VAR_INPUT CONSTANT PERSISTENT				
	fHys 					: REAL;				// constant light: hysteresis for control-deviation. Limited from 0 to rBrtns
	{attribute 'parameterUnit':= 'ms'}          
	nSwiOvrTi				: UDINT;			// distinction time [ms] between short click and long-press
	{attribute 'parameterUnit':= 's'}       	
	nSwiTi					: UDINT;			// switch-ramp-time [s] to drive rOut from 0 to 100 
	{attribute 'parameterUnit':= 's'}       	
	nDimTi					: UDINT;			// dim-ramp-time [s] to drive rOut from 0 to 100 
	{attribute 'parameterUnit':= 's'}       	
	nRampTi					: UDINT;			// constant light: control-ramp-time [s]
	{attribute 'parameterUnit':= 's'}           
	nPreOffRampTi			: UDINT;			// ramp time [s] for the pre-off-function
	{attribute 'parameterUnit':= 's'}       	
	nBrtnsAdjTi				: UDINT;			// constant light: time [s] to let the brighness sensor adjust to new values before taking them over to the internal control
	{attribute 'parameterUnit':= '%'}           
	fOnValCtrl				: REAL;				// on value in control mode, limited from 0 to 100.
	{attribute 'parameterUnit':= '%'}           
	fOnValMan				: REAL;				// on value in memory mode, limited from 0 to 100.
	{attribute 'parameterUnit':= '%'}           
	fPreOffVal				: REAL;				// light value on pre-off-delay period.
	{attribute 'parameterUnit':= 's'}           
	nPreOffDly				: UDINT;			// duration [s] of pre-off-delay period
	{attribute 'parameterUnit':= '%'}           
	fMinVal 				: REAL;				// constant light: minimum control-value before the light control wants to turn off
	{attribute 'parameterUnit':= 's'}           
	nMinOffDly 				: UDINT;			// constant light: time [s] before switching off at fMinVal
	{attribute 'parameterUnit':= 's'}           
	nMinOnDly 				: UDINT;			// constant light: time [s] before switching on at fMinVal
	bMemoryMode				: BOOL;				// memory mode. switch on to value before last off	
	{attribute 'parameterUnit':= 'KELVIN'}	                    
	fLgtT					: REAL		:= 3000;	
END_VAR	
		             
VAR_INPUT CONSTANT           	
	SpBrightness			: FB_BA_AV_Op;
	ManMode					: FB_BA_LightingEvt :=( ePrio:= E_BA_LightingPrio.eManual);	
	CnstLgtAuto				: FB_BA_LightingEvt :=( ePrio:= E_BA_LightingPrio.eAutomaticLight);
END_VAR
VAR
	ConstLgtCtrl			: FB_BA_LightCtrlConst;	
	PrioSwi					: FB_BA_LightingTgmSel4;	
END_VAR

// call of external control (e.g. HMI)
SUPER^(); // FB_BA_Ext_LightConstCtrl
SpBrightness(); // FB_BA_AV_Op
ConstLgtCtrl(
    bSwi := bManualSwitch,
    bSwiUp := FALSE,
    bSwiDwn := FALSE,
    bOn := bOn,
    bOff := bOff,
    fSetValMan := fSetLightValueMan_In,
    bSetValMan := bSetLightValueMan_In,
    bSetCtrlMod := bSetCtrlMod_In,
    bRstManMod := FALSE,
    bRst := bResetRoomFunction,
    bPrc := bPresence,
    fBrtns := fBrightness,
    fSP := SpBrightness.fPresentValue,
    fHys := fHys,
    nSwiOvrTi := nSwiOvrTi,
    nSwiTi := nSwiTi,
    nDimTi := nDimTi,
    nRampTi := nRampTi,
    nPreOffRampTi := nPreOffRampTi,
    nBrtnsAdjTi := nBrtnsAdjTi,
    fOnValCtrl := fOnValCtrl,
    fOnValMan := fOnValMan,
    fPreOffVal := fPreOffVal,
    nPreOffDly := nPreOffDly,
    fMinVal := fMinVal,
    nMinOffDly := nMinOffDly,
    nMinOnDly := nMinOnDly,
    bMemMod := bMemoryMode,
    eLgtActMod := eLightActivationMode_In,
    fRefLgtVal := stReferenceFeedback.fLightValue); // FB_BA_LightCtrlConst
CnstLgtAuto(bEn := ConstLgtCtrl.bControlMode, fLgtVal := ConstLgtCtrl.fOut, fLgtT := fLgtT); // FB_BA_LightingEvt
ManMode(bEn := ConstLgtCtrl.bManualMode, fLgtVal := ConstLgtCtrl.fOut, fLgtT := fLgtT); // FB_BA_LightingEvt
bAdjusting := ConstLgtCtrl.bAdjusting;
PrioSwi(
    stLightingTgm_1 := CnstLgtAuto.stLighting,
    stLightingTgm_2 := ManMode.stLighting,
    stLightingTgm_3 := stAreaLighting,
    stLightingTgm_4 := stScene); // FB_BA_LightingTgmSel4
stLighting := PrioSwi.stLighting;
eActualPrio_Out := PrioSwi.ePrioActvTgm;
fLightValue_Out := stReferenceFeedback.fLightValue;
// information to external control (e.g. HMI)
bLightOn_Out := stReferenceFeedback.fLightValue > 0;
bErr_Out := stReferenceFeedback.bErr;
bCtrlMod_Out := ConstLgtCtrl.bControlMode;
// Reset external control commands
bSetLightValueMan_In := FALSE;
bSetCtrlMod_In := FALSE;

METHOD FB_init : BOOL
VAR_INPUT
	bInitRetains : BOOL; // if TRUE, the retain variables are initialized (warm start / cold start)
	bInCopyCode : BOOL;  // if TRUE, the instance afterwards gets moved into the copy code (online change)
END_VAR
SpBrightness.iParent		:= THIS^;
SpBrightness.iLabel			:= LblFun_Setpoint;
SpBrightness.eUnit			:= E_BA_Unit.eLight_Luxes;  
SpBrightness.fValueRm		:= 300.0;
SpBrightness.fCOVIncrement	:= BA2_Param.fDefCOVIncrement;	

fHys 						:= 50;		// constant-light: hysteresis for control-deviation [lux].
nSwiOvrTi					:= 250;		// distinction-time [ms] between short-lick and long-press
nSwiTi						:= 2;		// switch-ramp-time [s] to drive rOut from 0 to 100 
nDimTi						:= 10;		// dim-ramp-time [s] to drive rOut from 0 to 100 
nRampTi						:= 60;		// constant-light: control-ramp-time [s]
nPreOffRampTi				:= 2;		// ramp-time [s] for the pre-off-function
nBrtnsAdjTi					:= 5;		// constant-light: time [s] to let the brighness-sensor adjust to new values before taking them over to the internal control
fOnValCtrl					:= 50;		// on-Value, limited from 0 to 100.
fOnValMan					:= 100;		// on-Value, limited from 0 to 100.
fPreOffVal					:= 4;		// light-value on pre-off-delay period.
nPreOffDly					:= 10;		// duration [s] of pre-off-delay period
fMinVal 					:= 4;		// constant-light: minimum control-value before the light control wants to turn off
nMinOffDly 					:= 300;		// constant-light: time [s] before switching off at fMinVal
nMinOnDly 					:= 300;		// constant-light: time [s] before switching on at fMinVal
bMemoryMode					:= FALSE;	// memory-mode. switch on to value before last off

fLgtT						:= 3000;			// [K]
END_METHOD

END_FUNCTION_BLOCK

// ---- Templates/POUs/Trade/RoomAutomation/Lighting/[Internal]/FB_BA_Ext_LightConstCtrl.TcPOU
{region '#Template'}
	{attribute 'Version' := '5.0.0.0'}
	{attribute 'Tags' := '"LCID": "1031", "Text": "RA, Beleuchtung, Anwenderfunktionen, Zone"'}
	{attribute 'Tags' := '"LCID": "1033", "Text": "RA, Lighting, User-functions, zone"'}
	{attribute 'Using' := '"Type": "Template", "URI": "ST_BA_LightActuatorFeedback"'}
	{attribute 'Description' := '"LCID": "1031", "Text": "Beleuchtung interner Baustein"'}
	{attribute 'Description' := '"LCID": "1033", "Text": "Lighting internal function"'}
{endregion}
FUNCTION_BLOCK FB_BA_Ext_LightConstCtrl EXTENDS FB_BA_Ext_LightCtrl
VAR	
	// data from/to user function
	{attribute 'BaParam.Title.DE' := 'Aktivieren Regelungsbetrieb'}
	{attribute 'BaParam.Title.EN' := 'Activate control mode'}
	{attribute 'BaParam.Access.Write' := 'Basic'}
	bSetCtrlMod_In				: BOOL;						// enter control mode from either deactivated or manual mode
	{attribute 'BaParam.Title.DE' := 'Regelungsbetrieb ist aktiv'}
	{attribute 'BaParam.Title.EN' := 'Control mode is active'}
	{attribute 'BaParam.Access.Write' := 'Locked'}
	{attribute 'BaParam.Access.Read' := 'Guest'}
	bCtrlMod_Out				: BOOL;						// state information control mode, used for external display
END_VAR

SUPER^();

END_FUNCTION_BLOCK

// ---- Templates/POUs/Trade/RoomAutomation/RoomSamples/FB_BA_RoomSample1.TcPOU
{region '#Template'}
	{attribute 'Version' := '6.0.0.0'}
	{attribute 'Tags' := '"LCID": "1031", "Text": "RA, Room, Sample"'}
	{attribute 'Tags' := '"LCID": "1033", "Text": "RA, Room, Sample"'}
	{attribute 'Using' := '"Type": "Template", "URI": "Site"'}
	{attribute 'Using' := '"Type": "Template", "URI": "BA2_Param"'}
	{attribute 'Using' := '"Type": "Template", "URI": "ST_BA_Facade"'}
	{attribute 'Using' := '"Type": "Template", "URI": "ST_BA_Lighting"'}
	{attribute 'Description' := '"LCID": "1031", "Text": "Beispiel Template Raum"'}
	{attribute 'Description' := '"LCID": "1033", "Text": "Sample-template room"'}
{endregion}
FUNCTION_BLOCK FB_BA_RoomSample1 EXTENDS FB_BA_View
VAR_INPUT
	stFacade					: ST_BA_Facade;			// sunblind-data from the next higher level
	stAreaLighting				: ST_BA_Lighting;		// lighting-data from the next higher level
END_VAR
		
VAR_INPUT CONSTANT PERSISTENT					
	{attribute 'parameterUnit':= 'KELVIN'}	                    
	fRmTAdjMin					: REAL;
	{attribute 'parameterUnit':= 'KELVIN'}	                    
	fRmTAdjMax					: REAL;
	{attribute 'parameterUnit':= 'KELVIN'}	                    
	fLgtT						: REAL;
	{attribute 'parameterUnit':= 's'}	                    
	nPollingIntervalFast		: UDINT;
	{attribute 'parameterUnit':= 's'}	                    
	nPollingIntervalNormal		: UDINT;
END_VAR	

VAR_INPUT CONSTANT
	BrtnsPrcSns					: FB_BA_BrightnessPresenceDALI;
	                    		
	Ctrl						: FB_BA_HeatCool_PID;
	VlvHtg						: FB_BA_ActuatorAnalog;
 	VlvCol						: FB_BA_ActuatorAnalog;
	                    		
	WdwCon1						: FB_BA_SensorBinary;
	WdwCon2						: FB_BA_SensorBinary;
	DewPointSensor				: FB_BA_SensorBinary;	
	RmTSen						: FB_BA_SensorAnalog;
	RmTAdj						: FB_BA_SensorAnalog;
	SunBldZone					: FB_BA_SunblindZone;
	SunBld1						: FB_BA_SunBld;		
	SunBld2						: FB_BA_SunBld;				
	LightZoneConstant			: FB_BA_LightGroupConstant;
	Light1						: FB_BA_LightAnalog;
	Light2						: FB_BA_LightAnalog;
END_VAR                 		
VAR                     		
	bSunbldSwiUp				: BOOL;
	bSunbldSwiDwn				: BOOL;	
	bLightSwi					: BOOL;	
	RmTAvg						: FB_BA_EnAvrg02;
	bInitializeSensor			: BOOL;	
END_VAR
VAR // added by the converter: edge detectors and wires of the graphical bodies
    _s1, _s2 : ST_BA_Analog;
END_VAR

SUPER^(); // FB_BA_View
BrtnsPrcSns(
    bEn := TRUE,
    bInitialize := bInitializeSensor,
    nPrdQueryBrtns := SEL(LightZoneConstant.bAdjusting, nPollingIntervalNormal, nPollingIntervalFast)); // FB_BA_BrightnessPresenceDALI
bInitializeSensor := FALSE;
WdwCon1(); // FB_BA_SensorBinary
WdwCon2(); // FB_BA_SensorBinary
DewPointSensor(); // FB_BA_SensorBinary
RmTSen(); // FB_BA_SensorAnalog
RmTAdj(); // FB_BA_SensorAnalog
Ctrl(
    bPrc := BrtnsPrcSns.bPresence,
    bWdwCon := NOT WdwCon1.bPresentValue OR NOT WdwCon2.bPresentValue,
    eMedium := Site.eHeatCoolMedium,
    bDewPnt := NOT DewPointSensor.bPresentValue,
    fRmT := RmTSen.fPresentValue,
    fRmTAdj := LIMIT(fRmTAdjMin, RmTAdj.fPresentValue, fRmTAdjMax),
    stBuildingSpRmT := Site.stBuildingSpRmT,
    eBuildingEnergyLevel := Site.eBuildingEnergyLevel); // FB_BA_HeatCool_PID
// compose _s1 : ST_BA_Analog
_s1.bEnPgm := Ctrl.bCtrlHtgActv;
_s1.fValPgm := Ctrl.fCtrlValHtg;
VlvHtg(stCmd := _s1); // FB_BA_ActuatorAnalog
// compose _s2 : ST_BA_Analog
_s2.bEnPgm := Ctrl.bCtrlColActv;
_s2.fValPgm := Ctrl.fCtrlValCol;
VlvCol(stCmd := _s2); // FB_BA_ActuatorAnalog
SunBldZone(
    fRoomTempSen := RmTAvg.fAvgVal,
    bPrcDetc := BrtnsPrcSns.bPresence,
    bSwiUp := bSunbldSwiUp,
    bSwiDwn := bSunbldSwiDwn,
    bRstManFnct := BrtnsPrcSns.bRstSwi,
    stBuildingSpRmT := Site.stBuildingSpRmT,
    stFacade := stFacade,
    stReferenceFeedback := SunBld1.stFeedback); // FB_BA_SunblindZone
SunBld2(bEn := TRUE, stSunBldCmd := SunBldZone.stSunBldOut); // FB_BA_SunBld
SunBld1(bEn := TRUE, stSunBldCmd := SunBldZone.stSunBldOut); // FB_BA_SunBld
LightZoneConstant(
    bManualSwitch := bLightSwi,
    bOn := FALSE,
    bOff := FALSE,
    bResetRoomFunction := BrtnsPrcSns.bRstSwi,
    bPresence := BrtnsPrcSns.bPresence,
    fBrightness := BrtnsPrcSns.fBrightness,
    stAreaLighting := stAreaLighting,
    stReferenceFeedback := Light1.stFeedback); // FB_BA_LightGroupConstant
Light2(bEn := TRUE, stLightingCmd := LightZoneConstant.stLighting); // FB_BA_LightAnalog
Light1(bEn := TRUE, stLightingCmd := LightZoneConstant.stLighting); // FB_BA_LightAnalog

METHOD FB_init : BOOL
VAR_INPUT
	bInitRetains : BOOL; // if TRUE, the retain variables are initialized (warm start / cold start)
	bInCopyCode : BOOL;  // if TRUE, the instance afterwards gets moved into the copy code (online change)
END_VAR
BrtnsPrcSns.iParent							:= THIS^;
BrtnsPrcSns.iLabel							:= LblCtl_BrightnessPresenceSensor; 			
BrtnsPrcSns.eDPADMode						:= E_BA_DPADMode.eInclude;	
BrtnsPrcSns.nAdr							:= 11;
BrtnsPrcSns.nInstancePresence				:= 1;	
BrtnsPrcSns.nInstanceBrightness				:= 0;
BrtnsPrcSns.nResBrtns						:= 10;
BrtnsPrcSns.ipDALICommunication				:= DALICommunication.fbKL6821Communication;

nPollingIntervalFast						:= 1;			// fast interval polling the light-value e.g. in case of active light-adapting
nPollingIntervalNormal						:= 15;			// slow interval polling the light-value

WdwCon1.iParent								:= THIS^;
WdwCon1.iLabel								:= LblAgg_WindowContact; 			
WdwCon1.eDPADMode							:= E_BA_DPADMode.eInclude;		
WdwCon1.Input.iLabel						:= LblFun_Status; 	
WdwCon1.Input.ePolarity						:= E_BA_Polarity.eReverse;
WdwCon1.Input.sActiveText 					:= txtEvent_Closed;
WdwCon1.Input.sInactiveText 				:= txtEvent_Opened;
WdwCon1.Input.nEventClassID					:= EC_ID.NC50;
WdwCon1.Input.aEventTransitionText[1]		:= txtEvent_Disturb;
WdwCon1.Input.aEventTransitionText[2]		:= txtEvent_None;
WdwCon1.Input.aEventTransitionText[3]		:= txtEvent_Normal;
WdwCon1.Input.bEventDetectionEnable			:= FALSE;
                                    		
WdwCon2.iParent								:= THIS^;
WdwCon2.iLabel								:= LblAgg_WindowContact; 			
WdwCon2.eDPADMode							:= E_BA_DPADMode.eInclude;		
WdwCon2.Input.iLabel						:= LblFun_Status; 	
WdwCon2.Input.ePolarity						:= E_BA_Polarity.eReverse;
WdwCon2.Input.sActiveText 					:= txtEvent_Closed;
WdwCon2.Input.sInactiveText 				:= txtEvent_Opened;
WdwCon2.Input.nEventClassID					:= EC_ID.NC50;
WdwCon2.Input.aEventTransitionText[1]		:= txtEvent_Disturb;
WdwCon2.Input.aEventTransitionText[2]		:= txtEvent_None;
WdwCon2.Input.aEventTransitionText[3]		:= txtEvent_Normal;
WdwCon2.Input.bEventDetectionEnable			:= FALSE;

DewPointSensor.iParent						:= THIS^;
DewPointSensor.iLabel						:= LblAgg_MonitorDewPoint; 			
DewPointSensor.eDPADMode					:= E_BA_DPADMode.eInclude;		
DewPointSensor.Input.iLabel					:= LblFun_Status; 	
DewPointSensor.Input.ePolarity				:= E_BA_Polarity.eReverse;	
DewPointSensor.Input.sActiveText 			:= txtEvent_Normal;
DewPointSensor.Input.sInactiveText 			:= txtEvent_Triggered;
DewPointSensor.Input.nEventClassID			:= EC_ID.NC40;
DewPointSensor.Input.aEventTransitionText[1]:= txtEvent_Triggered;
DewPointSensor.Input.aEventTransitionText[2]:= txtEvent_None;
DewPointSensor.Input.aEventTransitionText[3]:= txtEvent_Normal;
DewPointSensor.Input.bEventDetectionEnable	:= TRUE;

RmTSen.iParent								:= THIS^;
RmTSen.iLabel								:= LblAgg_TemperatureRoomAir; 			
RmTSen.eDPADMode							:= E_BA_DPADMode.eInclude;		
RmTSen.MV.eUnit 							:= E_BA_Unit.eTemperature_DegreesCelsius;
RmTSen.MV.nEventClassID						:= EC_ID.NC60;
RmTSen.MV.aEventTransitionText[1]			:= txtEvent_Disturb;
RmTSen.MV.aEventTransitionText[2]			:= txtEvent_None;
RmTSen.MV.aEventTransitionText[3]			:= txtEvent_Normal;
RmTSen.MV.eEnPlantLock						:= E_BA_LockPriority.eNoLock;
RmTSen.MV.fResolution 						:= 0.01;
RmTSen.MV.fScaleOffset 						:= 0; 
                     			        	
RmTAdj.iParent								:= THIS^;
RmTAdj.iLabel								:= LblAgg_RoomControlUnit; 	
RmTAdj.eDPADMode							:= E_BA_DPADMode.eInclude;		
RmTAdj.MV.eUnit 							:= E_BA_Unit.eTemperature_DegreesKelvin;
RmTAdj.MV.nEventClassID						:= EC_ID.NC60;
RmTAdj.MV.aEventTransitionText[1]			:= txtEvent_Disturb;
RmTAdj.MV.aEventTransitionText[2]			:= txtEvent_None;
RmTAdj.MV.aEventTransitionText[3]			:= txtEvent_Normal;
RmTAdj.MV.eEnPlantLock						:= E_BA_LockPriority.eNoLock;
RmTAdj.MV.fResolution 						:= 0.01;
RmTAdj.MV.fScaleOffset 						:= 0; 
        
fRmTAdjMin									:= -5;	// limits of room-temperature-adjustment           
fRmTAdjMax									:= 5;	// in order to prevent adjusting from 0 to 50 degrees, for example

Ctrl.iParent								:= THIS^;
Ctrl.iLabel									:= LblCtl_RoomTemperatureControl; 			 
Ctrl.eDPADMode								:= E_BA_DPADMode.eInclude;

VlvHtg.iParent								:= THIS^;
VlvHtg.iLabel								:= LblAgg_Valve; 	
VlvHtg.eDPADMode							:= E_BA_DPADMode.eInclude;
VlvHtg.Mdlt.eUnit 							:= E_BA_Unit.eOther_Percent;
VlvHtg.Mdlt.nEventClassID					:= EC_ID.NC60;
VlvHtg.Mdlt.aEventTransitionText[1]			:= txtEvent_Disturb;
VlvHtg.Mdlt.aEventTransitionText[2]			:= txtEvent_None;
VlvHtg.Mdlt.aEventTransitionText[3]			:= txtEvent_Normal;		
VlvHtg.Mdlt.fResolution 					:= 0.01;
VlvHtg.Mdlt.fScaleOffset 					:= 0; 		 
                            			    
VlvCol.iParent								:= THIS^;
VlvCol.iLabel								:= LblAgg_Valve; 	
VlvCol.eDPADMode							:= E_BA_DPADMode.eInclude;
VlvCol.Mdlt.eUnit 							:= E_BA_Unit.eOther_Percent;
VlvCol.Mdlt.nEventClassID					:= EC_ID.NC60;
VlvCol.Mdlt.aEventTransitionText[1]			:= txtEvent_Disturb;
VlvCol.Mdlt.aEventTransitionText[2]			:= txtEvent_None;
VlvCol.Mdlt.aEventTransitionText[3]			:= txtEvent_Normal;		
VlvCol.Mdlt.fResolution 					:= 0.01;
VlvCol.Mdlt.fScaleOffset 					:= 0; 



SunBldZone.iParent							:= THIS^;
SunBldZone.iLabel							:= LblCtl_SunblindZoneControl; 		

Sunbld1.iParent								:= THIS^;
Sunbld1.iLabel								:= LblCtl_SunblindActuator; 	
Sunbld1.sObjectName							:= '{Idx=01}';		 		 
Sunbld1.eDPADMode							:= E_BA_DPADMode.eInclude;

Sunbld2.iParent								:= THIS^;
Sunbld2.iLabel								:= LblCtl_SunblindActuator; 	
Sunbld2.sObjectName							:= '{Idx=02}';	 		 
Sunbld2.eDPADMode							:= E_BA_DPADMode.eInclude;



Light1.iParent								:= THIS^;
Light1.iLabel								:= LblCtl_LightActuator; 	
Light1.sObjectName							:= '{Idx=01}';		 
Light1.eDPADMode							:= E_BA_DPADMode.eInclude;

Light2.iParent								:= THIS^;
Light2.iLabel								:= LblCtl_LightActuator; 		
Light2.sObjectName							:= '{Idx=02}';	 
Light2.eDPADMode							:= E_BA_DPADMode.eInclude;

LightZoneConstant.iParent					:= THIS^;
LightZoneConstant.iLabel					:= LblCtl_LightZoneControl; 			 
LightZoneConstant.eDPADMode					:= E_BA_DPADMode.eInclude;

fLgtT										:= 3000;		// light-temperature [K]
END_METHOD

END_FUNCTION_BLOCK

// ---- Templates/POUs/Trade/RoomAutomation/SunProtection/Actuators/FB_BA_SunBld.TcPOU
{region '#Template'}
	{attribute 'Version' := '6.0.0.0'}
	{attribute 'Tags' := '"LCID": "1031", "Text": "RA, Sunprotection, Sunblind"'}
	{attribute 'Tags' := '"LCID": "1033", "Text": "RA, Sunprotection, Sunblind"'}
	{attribute 'Using' := '"Type": "Template", "URI": "BA2_Param"'}
	{attribute 'Using' := '"Type": "Template", "URI": "ST_BA_SunblindActuatorFeedback"'}
	{attribute 'Description' := '"LCID": "1031", "Text": "Sonnenschutzaktor (Jalousie)"'}
	{attribute 'Description' := '"LCID": "1033", "Text": "Sunblind-actuator (venetian blind)"'}
{endregion}
FUNCTION_BLOCK FB_BA_SunBld EXTENDS FB_BA_View


VAR_INPUT
	bEn						: BOOL;
	stSunBldCmd				: ST_BA_SunBld;		// Low-Priorities command telegram
END_VAR
VAR_OUTPUT
	bReferencing			: BOOL;				// device is being referenced
	nReferenceTimer			: UDINT;            
	bErr					: BOOL;				// error
	fActualPosition			: REAL;				// actual position
	fActualAngle			: REAL;				// actual angle
	eActualSunblindPrio		: BYTE;				// actual telegram priority
	stFeedback				: ST_BA_SunblindActuatorFeedback;
END_VAR
VAR_INPUT CONSTANT PERSISTENT
	{attribute 'parameterUnit':= 'ms'}
	nPositioningDelay		: UDINT;	// delay of automatic telegrams [ms] to prevent overload
	{attribute 'parameterUnit':= 'ms'}  
	nTiUp					: UDINT;	// total driving-up-time [ms]
	{attribute 'parameterUnit':= 'ms'}  
	nTiDwn					: UDINT;	// total driving-down-time [ms]
	{attribute 'parameterUnit':= 'ms'}          		
	nTurnTiUp				: UDINT;	// time to turn lamellas up [ms]
	{attribute 'parameterUnit':= 'ms'}          		
	nTurnTiDwn				: UDINT;	// time to turn lamellas down [ms]
	{attribute 'parameterUnit':= 'ms'}          		
	nBckLshTiUp				: UDINT;	// Time to traverse the backlash in the upward direction [ms]
	{attribute 'parameterUnit':= 'ms'}          		
	nBckLshTiDwn			: UDINT;	// Time to traverse the backlash in the downward direction [ms]
	{attribute 'parameterUnit':= 'deg'} 
	fAnglLmtUp				: REAL;		// upper limit of lamellas in deg - must be greater than fAnglLmtDwn
	{attribute 'parameterUnit':= 'deg'} 
	fAnglLmtDwn				: REAL;		// lower limit of lamellas in deg - must be lower than fAnglLmtUp
END_VAR
VAR_INPUT CONSTANT				 
	ActualPosition			: FB_BA_AV_Op;		
	ActualAngle				: FB_BA_AV_Op;		
END_VAR
VAR
	PositioningDelay		: FB_BA_SunBldPosDly;
	SunBldActr				: FB_BA_SunBldActr;
	bCmdUp			AT %Q*	: BOOL;
	bCmdDown		AT %Q*	: BOOL;
END_VAR
VAR // added by the converter: edge detectors and wires of the graphical bodies
    _s1 : ST_BA_SunblindActuatorFeedback;
END_VAR

SUPER^(); // FB_BA_View
PositioningDelay(stIn := stSunBldCmd, nDly := nPositioningDelay); // FB_BA_SunBldPosDly
SunBldActr(
    bEn := bEn,
    stCmd := PositioningDelay.stOut,
    nTiUp := nTiUp,
    nTiDwn := nTiDwn,
    nTurnTiUp := nTurnTiUp,
    nTurnTiDwn := nTurnTiDwn,
    nBckLshTiUp := nBckLshTiUp,
    nBckLshTiDwn := nBckLshTiDwn,
    fAnglLmtUp := fAnglLmtUp,
    fAnglLmtDwn := fAnglLmtDwn); // FB_BA_SunBldActr
bCmdUp := SunBldActr.bUp;
bCmdDown := SunBldActr.bDwn;
fActualPosition := SunBldActr.fActlPos;
fActualAngle := SunBldActr.fActlAngl;
bReferencing := SunBldActr.bRef;
nReferenceTimer := SunBldActr.nRefTi;
bErr := SunBldActr.bErr;
ActualPosition(fValuePgm := fActualPosition); // FB_BA_AV_Op
ActualAngle(fValuePgm := fActualAngle); // FB_BA_AV_Op
eActualSunblindPrio := stSunBldCmd.ePrio;
// compose _s1 : ST_BA_SunblindActuatorFeedback
_s1.bReferencing := SunBldActr.bRef;
_s1.bErr := SunBldActr.bErr;
_s1.bBusy := SunBldActr.bBusy;
_s1.ePrio := stSunBldCmd.ePrio;
_s1.fPosition := SunBldActr.fActlPos;
_s1.fAngle := SunBldActr.fActlAngl;
_s1.fAnglLmtUp := fAnglLmtUp;
_s1.fAnglLmtDwn := fAnglLmtDwn;
stFeedback := _s1;

METHOD FB_init : BOOL
VAR_INPUT
	bInitRetains : BOOL; // if TRUE; the retain variables are initialized (warm start / cold start)
	bInCopyCode : BOOL;  // if TRUE; the instance afterwards gets moved into the copy code (online change)
END_VAR
nPositioningDelay				:= 250;			// delay of automatic telegrams [ms] to prevent overload
nTiUp							:= 50000;		// total driving-up-time [ms]
nTiDwn							:= 50000;		// total driving-down-time [ms]
nTurnTiUp						:= 1500;		// time to turn lamellas up [ms]
nTurnTiDwn						:= 1500;		// time to turn lamellas down [ms]
nBckLshTiUp						:= 100;			// Time to traverse the backlash in the upward direction [ms]
nBckLshTiDwn					:= 100;			// Time to traverse the backlash in the downward direction [ms]
fAnglLmtUp						:= 30;			// upper limit of lamellas in deg - must be greater than fAnglLmtDwn
fAnglLmtDwn						:= -70;			// lower limit of lamellas in deg - must be lower than fAnglLmtUp

// actual position / aktueller Position
ActualPosition.iParent			:= THIS^;
ActualPosition.iLabel			:= LblFun_FeedbackSunblindPosition;
ActualPosition.eUnit			:= E_BA_Unit.eOther_Percent;
ActualPosition.fCOVIncrement	:= BA2_Param.fDefCOVIncrement;

// actual angle / aktueller Lamellenwinkel
ActualAngle.iParent				:= THIS^;
ActualAngle.iLabel				:= LblFun_FeedbackSunblindAngle;
ActualAngle.eUnit				:= E_BA_Unit.eOther_DegreesAngular;
ActualAngle.fCOVIncrement		:= BA2_Param.fDefCOVIncrement;
END_METHOD

END_FUNCTION_BLOCK

// ---- Templates/POUs/Trade/RoomAutomation/SunProtection/[Internal]/FB_BA_Ext_SunblindBase.TcPOU
{region '#Template'}
	{attribute 'Version' := '5.0.0.0'}
	{attribute 'Tags' := '"LCID": "1031", "Text": "RA, Sunprotection, Sunblind, Zone"'}
	{attribute 'Tags' := '"LCID": "1033", "Text": "RA, Sunprotection, Sunblind, Zone"'}
	{attribute 'Using' := '"Type": "Template", "URI": "ST_BA_Facade"'}
	{attribute 'Description' := '"LCID": "1031", "Text": "Sonnenschutzlogik interner Baustein"'}
	{attribute 'Description' := '"LCID": "1033", "Text": "Sunblind-logic inernal function)"'}
{endregion}
FUNCTION_BLOCK FB_BA_Ext_SunblindBase EXTENDS FB_BA_Object
VAR_INPUT
	bRstManFnct				: BOOL;								// reset the external function from outside
END_VAR
VAR		
	{attribute 'BaParam.Title.DE' := 'Hoch'}
	{attribute 'BaParam.Title.EN' := 'Up'}
	{attribute 'BaParam.Access.Write' := 'Basic'}
	bUp_In					: BOOL;								// from external
	{attribute 'BaParam.Title.DE' := 'Herunter'}
	{attribute 'BaParam.Title.EN' := 'Down'}
	{attribute 'BaParam.Access.Write' := 'Basic'}
	bDown_In				: BOOL;								// from external
	{attribute 'BaParam.Title.DE' := 'Reset Hand'}
	{attribute 'BaParam.Title.EN' := 'Reset manual'}
	{attribute 'BaParam.Access.Write' := 'Basic'}
	bResetManual_In			: BOOL;								// from external
	{attribute 'BaParam.Title.DE' := 'Rückmeldung Fehler'}
	{attribute 'BaParam.Title.EN' := 'Feedback Error'}
	{attribute 'BaParam.Access.Write' := 'Locked'}
	{attribute 'BaParam.Access.Read' := 'Guest'}
	bErr_Out				: BOOL;								// to external
	{attribute 'BaParam.Title.DE' := 'Rückmeldung geöffnet'}
	{attribute 'BaParam.Title.EN' := 'Feedback open'}
	{attribute 'BaParam.Access.Write' := 'Locked'}
	{attribute 'BaParam.Access.Read' := 'Guest'}
	bOpened_Out				: BOOL;								// to external
	{attribute 'BaParam.Title.DE' := 'Rückmeldung geschlossen'}
	{attribute 'BaParam.Title.EN' := 'Feedback close'}
	{attribute 'BaParam.Access.Write' := 'Locked'}
	{attribute 'BaParam.Access.Read' := 'Guest'}
	bClosed_Out				: BOOL;								// to external
	{attribute 'BaParam.Title.DE' := 'Aktuell steuernde Priorität'}
	{attribute 'BaParam.Title.EN' := 'Actual controlling priority'}
	{attribute 'BaParam.Access.Write' := 'Locked'}
	{attribute 'BaParam.Access.Read' := 'Guest'}
	eActualPrio_Out			: BYTE;								// priority of resulting zone-telegram
		                                                    	
	                                                        	
	bInitialize_In			: BOOL;								// from external // actually not used by external control
	bBusy					: BOOL;								// to external // actually not used by external control
	bReferencing			: BOOL;								// to external // actually not used by external control
	bBlindMoving			: BOOL;                         	
	                                                        	
	stSunblindCmdExt		: ST_BA_SunBld;						// telegram assembled from external data
	stSunblindCmdResult		: ST_BA_SunBld;						// telegram to extract information for external handling
		                    
	rtUp					: R_TRIG;
	rtDown					: R_TRIG;
	rtReferencing			: R_TRIG;
	ftBusy					: F_TRIG;
	                        
	_nResetManual_In		: BYTE;
	_nInitialize_In			: BYTE;
END_VAR
VAR_INPUT CONSTANT PERSISTENT
	ePrio					: BYTE	:= E_BA_SunbldPrio.eManualGroup;	// priority of external telegram
END_VAR

SUPER^();

// predefinition of priority
stSunblindCmdExt.ePrio		:= ePrio;

// state moving
bBlindMoving	:= bBusy AND NOT bReferencing;

// reset telegram from outside or from HMI or set 0%/100% as on/off
IF bRstManFnct	OR (bResetManual_In AND (_nResetManual_In=1))	THEN	// bResetManual_In has to go through the other parts first before having an effect here
	stSunblindCmdExt.bActv			:= FALSE;
	stSunblindCmdExt.bManUp			:= FALSE;
	stSunblindCmdExt.bManDwn		:= FALSE;
	stSunblindCmdExt.bManMod		:= FALSE;
ELSIF (bUp_In OR bDown_In) AND_THEN bBlindMoving	THEN   		// stop while driving
		stSunblindCmdExt.bManUp		:= FALSE; 
		stSunblindCmdExt.bManDwn	:= FALSE;
ELSIF bUp_In								THEN    
		stSunblindCmdExt.bManUp		:= TRUE;
		stSunblindCmdExt.bManDwn	:= FALSE;
ELSIF bDown_In 							THEN   
		stSunblindCmdExt.bManUp		:= FALSE; 
		stSunblindCmdExt.bManDwn	:= TRUE;
END_IF

IF	bOpened_Out	THEN    
		stSunblindCmdExt.bManUp		:= FALSE;
END_IF
IF	bClosed_Out	THEN    
		stSunblindCmdExt.bManDwn	:= FALSE;
END_IF

rtUp	(CLK:=	stSunblindCmdExt.bManUp);
rtDown	(CLK:=	stSunblindCmdExt.bManDwn);

IF rtUp.Q	OR rtDown.Q	THEN
	stSunblindCmdExt.bActv			:= TRUE;
	stSunblindCmdExt.bManMod		:= TRUE;
	// Event-increment as timestamp
	BA_Globals.nEvtIncSunBld		:= BA_Globals.nEvtIncSunBld+1;
	stSunblindCmdExt.nEvtInc		:= BA_Globals.nEvtIncSunBld;
END_IF

ftBusy			(CLK := bBusy);			// trigger for children to take over the actual values as target-values
rtReferencing	(CLK := bReferencing);	// trigger for children to take over the actual values as target-values
bUp_In	:= bDown_In	:= FALSE;

// reset bResetManual_In after one cycle
IF bResetManual_In	THEN
	_nResetManual_In	:= _nResetManual_In+1;
	IF _nResetManual_In>=2	THEN
		bResetManual_In	:= FALSE;
		_nResetManual_In	:= 0;
	END_IF
END_IF

// reset bInitialize_In after one cycle
IF bInitialize_In	THEN
	_nInitialize_In	:= _nInitialize_In+1;
	IF _nInitialize_In>=2	THEN
		bInitialize_In	:= FALSE;
		_nInitialize_In	:= 0;
	END_IF
END_IF

END_FUNCTION_BLOCK

// ---- Templates/POUs/Universal/Control/Scale/FB_BA_Scale_04.TcPOU
{region '#Template'}
	{attribute 'Version' := '5.0.0.0'}
	{attribute 'Tags' := '"LCID": "1031", "Text": "Universal, Control, Scaling"'}
	{attribute 'Tags' := '"LCID": "1033", "Text": "Universal, Control, Scaling"'}
	{attribute 'Using' := '"Type": "Template", "URI": "BA2_Param"'}
	{attribute 'Description' := '"LCID": "1031", "Text": "Skalierung"'}
	{attribute 'Description' := '"LCID": "1033", "Text": "Scaling"'}
{endregion}
FUNCTION_BLOCK FB_BA_Scale_04 EXTENDS FB_BA_View
VAR_INPUT
	fX			: REAL;
END_VAR
VAR_OUTPUT
	fY			: REAL;
END_VAR
VAR_INPUT CONSTANT
	X1			: FB_BA_AV_Op;	
	X2			: FB_BA_AV_Op;	
	X3			: FB_BA_AV_Op;	
	X4			: FB_BA_AV_Op;	
	Y1			: FB_BA_AV_Op;	
	Y2			: FB_BA_AV_Op;
	Y3			: FB_BA_AV_Op;
	Y4			: FB_BA_AV_Op;
	YMin		: FB_BA_AV_Op;			
	YMax		: FB_BA_AV_Op;			
	Y			: FB_BA_AV_Op;		
END_VAR
VAR		
	Scale		: FB_BA_Chrct04;
END_VAR

SUPER^(); // FB_BA_View
X1(); // FB_BA_AV_Op
X2(); // FB_BA_AV_Op
X3(); // FB_BA_AV_Op
X4(); // FB_BA_AV_Op
Y1(); // FB_BA_AV_Op
Y2(); // FB_BA_AV_Op
Y3(); // FB_BA_AV_Op
Y4(); // FB_BA_AV_Op
Ymin(); // FB_BA_AV_Op
YMax(); // FB_BA_AV_Op
Scale(
    fX := fX,
    fX01 := X1.fPresentValue,
    fX02 := X2.fPresentValue,
    fX03 := X3.fPresentValue,
    fX04 := X4.fPresentValue,
    fY01 := Y1.fPresentValue,
    fY02 := Y2.fPresentValue,
    fY03 := Y3.fPresentValue,
    fY04 := Y4.fPresentValue,
    fYMin := Ymin.fPresentValue,
    fYMax := YMax.fPresentValue); // FB_BA_Chrct04
Y(fValuePgm := Scale.fCalcVal); // FB_BA_AV_Op
fY := Y.fPresentValue;

METHOD FB_init : BOOL
VAR_INPUT
	bInitRetains : BOOL; // if TRUE, the retain variables are initialized (warm start / cold start)
	bInCopyCode : BOOL;  // if TRUE, the instance afterwards gets moved into the copy code (online change)
END_VAR
X1.iParent			:= THIS^;
X1.iLabel		:= LblCtl_X01;  							 	 
X1.eUnit			:= E_BA_Unit.eTemperature_DegreesCelsius;						 	 
X1.fValueRm			:= 15.0;
X1.fCOVIncrement	:= BA2_Param.fDefCOVIncrement;		

X2.iParent			:= THIS^;
X2.iLabel		:= LblCtl_X02;  								 	 
X2.eUnit			:= E_BA_Unit.eTemperature_DegreesCelsius;						 	 
X2.fValueRm			:= 0.0;
X2.fCOVIncrement	:= BA2_Param.fDefCOVIncrement;		

X3.iParent			:= THIS^;
X3.iLabel		:= LblCtl_X03;  								 	 
X3.eUnit			:= E_BA_Unit.eTemperature_DegreesCelsius;						 	 
X3.fValueRm			:= -20.0;
X3.fCOVIncrement	:= BA2_Param.fDefCOVIncrement;			

X4.iParent			:= THIS^;
X4.iLabel		:= LblCtl_X04;  									 	 
X4.eUnit			:= E_BA_Unit.eTemperature_DegreesCelsius;						 	 
X4.fValueRm			:= -20.0;
X4.fCOVIncrement	:= BA2_Param.fDefCOVIncrement;		

Y1.iParent			:= THIS^;
Y1.iLabel		:= LblCtl_Y01;  			 	 
Y1.eUnit			:= E_BA_Unit.eTemperature_DegreesCelsius;						 	 
Y1.fValueRm			:= 25.0;
Y1.fCOVIncrement	:= BA2_Param.fDefCOVIncrement;		

Y2.iParent			:= THIS^;
Y2.iLabel		:= LblCtl_Y02;  							 	 
Y2.eUnit			:= E_BA_Unit.eTemperature_DegreesCelsius;						 	 
Y2.fValueRm			:= 40.0;
Y2.fCOVIncrement	:= BA2_Param.fDefCOVIncrement;		

Y3.iParent			:= THIS^;
Y3.iLabel			:= LblCtl_Y03;  							 	 
Y3.eUnit			:= E_BA_Unit.eTemperature_DegreesCelsius;						 	 
Y3.fValueRm			:= 60.0;
Y3.fCOVIncrement	:= BA2_Param.fDefCOVIncrement;		


Y4.iParent			:= THIS^;
Y4.iLabel			:= LblCtl_Y04;  									 	 
Y4.eUnit			:= E_BA_Unit.eTemperature_DegreesCelsius;						 	 
Y4.fValueRm			:= 65.0;
Y4.fCOVIncrement	:= BA2_Param.fDefCOVIncrement;		

YMin.iParent		:= THIS^;
YMin.iLabel			:= LblFun_MinimumValue;										 	 
YMin.eUnit			:= E_BA_Unit.eTemperature_DegreesCelsius;						 	 
YMin.fValueRm		:= 5.0;
YMin.fCOVIncrement	:= BA2_Param.fDefCOVIncrement;		

YMax.iParent		:= THIS^;
YMax.iLabel			:= LblFun_MaximumValue;							 	 
YMax.eUnit			:= E_BA_Unit.eTemperature_DegreesCelsius;						 	 
YMax.fValueRm		:= 80.0;
YMax.fCOVIncrement	:= BA2_Param.fDefCOVIncrement;		

Y.iParent			:= THIS^;
Y.iLabel			:= LblFun_SetpointCalculated;										 	 
Y.eUnit				:= E_BA_Unit.eTemperature_DegreesCelsius;	
Y.fCOVIncrement		:= BA2_Param.fDefCOVIncrement;
END_METHOD

END_FUNCTION_BLOCK

// ---- Templates/POUs/Universal/Control/TimeDelay/FB_BA_DlyOn.TcPOU
{region '#Template'}
	{attribute 'Version' := '5.0.0.0'}
	{attribute 'Tags' := '"LCID": "1031", "Text": "Universal, Control, Timer"'}
	{attribute 'Tags' := '"LCID": "1033", "Text": "Universal, Control, Timer"'}
	{attribute 'Using' := '"Type": "Template", "URI": "BA2_Param"'}
	{attribute 'Description' := '"LCID": "1031", "Text": "Zeitglied Einschaltverzögert"'}
	{attribute 'Description' := '"LCID": "1033", "Text": "Timer switch-on delayed"'}
{endregion}
FUNCTION_BLOCK FB_BA_DlyOn EXTENDS FB_BA_View
VAR_INPUT
	bVal					: BOOL;	
END_VAR
VAR_OUTPUT
	bQ						: BOOL;
	nRT						: UDINT;// Restzeit [s] // remaining time [s]	
END_VAR
VAR_INPUT CONSTANT
	TiDly					: FB_BA_AV_Op;		
END_VAR	
VAR	
	tonDlyOn				: TON;
END_VAR
VAR // added by the converter: edge detectors and wires of the graphical bodies
    _w1, _w2 : ANY;
END_VAR

SUPER^(); // FB_BA_View
TiDly(); // FB_BA_AV_Op
_w1 := F_BA_RealToTiSec(fSec := TiDly.fPresentValue);
tonDlyOn(IN := bVal, PT := _w1); // TON
bQ := tonDlyOn.Q;
_w2 := F_BA_RemSecsTon(tonTimer := tonDlyOn);
nRT := _w2;

METHOD FB_init : BOOL
VAR_INPUT
	bInitRetains : BOOL; // if TRUE, the retain variables are initialized (warm start / cold start)
	bInCopyCode : BOOL;  // if TRUE, the instance afterwards gets moved into the copy code (online change)
END_VAR
TiDly.iParent			:= THIS^; 
TiDly.iLabel			:= LblCtl_TimeDelay;
TiDly.eUnit 			:= E_BA_Unit.eTime_Seconds;								 
TiDly.fValueRm			:= 0;		
TiDly.fCOVIncrement		:= BA2_Param.fDefCOVIncrement;
END_METHOD

END_FUNCTION_BLOCK
